FUNCTION_BLOCK FB_WeatherStation
VAR_INPUT
END_VAR
VAR_OUTPUT
END_VAR
VAR
END_VAR

END_FUNCTION_BLOCK

(* stored: Version 1.1.0.1, ProductVersion 3.1.4024.10
   POU FB_WeatherStation: Id {2223274a-fac9-415f-ac72-babfc7b551f4}, SpecialFunc None *)
